{attribute 'qualified_only'}
VAR_GLOBAL
	// ================= Tool Types ====================================
	//TODO: change 
	quarterInchUpcut : Tool_Type := (speed := 18000, toolNumber := 2, modelname := 'Dimar', name := 'Quarter Inch Upcut', x_coord := 1, y_coord := 122, z_coord := 441);
	halfInchUpcut : Tool_Type := (speed := 22000, toolNumber := 4, modelname := 'Dimar', name := 'Half Inch Upcut', x_coord := 0, y_coord := 132, z_coord := 452);
	sawblade : Tool_Type := (speed := 10000, toolNumber := 0, modelname := 'Hunter Precision Tools', name := 'Sawblade', x_coord := 71, y_coord := 193, z_coord := 509);
	dovetail : Tool_Type := (speed := 18000, toolNumber := 5, modelname := 'Dimar', name := 'Dovetail');
	halfInchBall : Tool_Type := (speed := 18000, toolNumber := 6, modelname := 'Dimar', name := 'Half Inch Ball');
//	quarterInchBall : Tool_Type := (speed := 18000, toolNumber := 7, modelname := 'Dimar', name := 'Quarter Inch Ball');
	noTool : Tool_Type := (speed := 0, toolNumber := 8, modelname := 'Dimar', name := 'None');

	// ================= Programs ====================================
	//Update C:\Users\kris\OneDrive\Documents\Robot transfer\Robot Programs\BX130XControlCode\BX130XControlCode\BX130XPLC\POUs\FB_Machine.TcPOU
	FrontWall : Program_Type := (index := 1, option1true := 'E cut', option1false := 'No E cut', option2true := 'Glass Door', option2false := 'Standard Door', option3true := 'Handles', option3false := 'No Handles', programName := 'Front Wall', firstTool := halfInchUpcut);
	BackWall : Program_Type := (index := 2, option1true := 'XL Window', option1false := 'No Window', option2true := 'Handles', option2false := 'No Handles', option3true := 'Glass Door Handle', option3false := 'No Glass Door Handle', programName := 'Back Wall', firstTool := halfInchUpcut);	
	Option3 : Program_Type := (index := 3, option1true := 'Rear Wall', option1false := 'Front Wall', option2true := '', option2false := '', option3true := '', option3false := '', programName := 'Cube Blade Only', firstTool := quarterInchUpcut);
	Option4 : Program_Type := (index := 4, option1true := '', option1false := '', option2true := '', option2false := '', option3true := '', option3false := '', programName := 'Option4', firstTool := quarterInchUpcut);
	CubeSaunaFront : Program_Type := (index := 5, option1true := 'Rear Wall', option1false := 'Front Wall', option2true := 'Glass Door', option2false := 'Standard Door', option3true := 'Blade Only', option3false := 'Not Blade Only', programName := 'Cube Sauna', firstTool := halfInchUpcut);
	Option5 : Program_Type := (index := 6, option1true := 'Glass Door Front', option1false := '', option2true := 'Wood Door Front', option2false := '', option3true := 'XL Window Rear', option3false := '', programName := 'option5', firstTool := halfInchUpcut);
	Option6 : Program_Type := (index := 7, option1true := '', option1false := '', option2true := '', option2false := '', option3true := '', option3false := '', programName := 'Wings Only', firstTool := halfInchUpcut);
	Option7 : Program_Type := (index := 8, option1true := '', option1false := '', option2true := '', option2false := '', option3true := '', option3false := '', programName := 'option7', firstTool := halfInchUpcut);
	CubeSaunaRear : Program_Type := (index := 9, option1true := '', option1false := '', option2true := '', option2false := '', option3true := '', option3false := '', programName := 'CubeSaunaRear', firstTool := halfInchUpcut);
	ToolChange : Program_Type := (index := 10, option1true := '', option1false := '', option2true := '', option2false := '', option3true := '', option3false := '', programName := 'ToolChange', firstTool := quarterInchUpcut);

	//=============== Constants ===
	calibrationPlasticZHeight : REAL := 493.3;
END_VAR

(* stored: Version 1.1.0.1, ProductVersion 3.1.4024.12
   GVL GVL_Programs: Id {1d7e22d7-5577-4dde-a98e-416112e79629} *)
